(*********************************** G.D S.p.A. - Technical Department ***********************************
============= PROGRAM INFO ============
FOLDER:             TBD
MACHINES INVOLVED:  TBD 

============= DESCRIPTION =============

============= REVISIONS ===============
Date		Version	 	Author      	Description             
----------	-------		------------  	--------------------------------------------
2019/04/24 	0000.00	 	M.Grasso		Creation of the PRG

**********************************************************************************************************)
(*$R
	process_ref := prc;
$*)
PROGRAM csp_main_safety
VAR
	prc:					process;
	prc_path:				STRING;
	
	series_closed_dvr:		BOOL;
	
END_VAR

_read_var_input();

_object_manager();

IF NOT objects_running()
THEN
	RETURN;	
END_IF

_read_process_image();

_mode_manager();

CASE process_get_mode(prc) of
	MODE_ABSENT,
	MODE_INACTIVE:
		RETURN;
	MODE_TEST:
		_handle_process_test();
END_CASE

_set_runtime_properties();

(********************************* BODY *********************************)

(************************************************************************)

_handle_messages();

_write_output();

ACTION _handle_messages:
;
END_ACTION

ACTION _handle_process_test:
;
END_ACTION

ACTION _mode_manager:
IF process_mode_req_is_pending(prc)
THEN
    process_apply_mode_req_first_step(prc);
    CASE process_get_mode(prc) OF
        MODE_TO_ABSENT:
			;
        MODE_TO_INACTIVE:
			;
        MODE_TO_TEST:
			;
        MODE_TO_OPERATIONAL:
			;
    END_CASE
    process_apply_mode_req_second_step(prc);
END_IF
END_ACTION

ACTION _object_manager:
IF objects_initialization()
THEN
	sub_process_init(
		object_name					:= 'csp_main_safety.prc', 
		process						:= csp_main.prc, 
		CONVERSION_this				:= prc);
		
	prc_path 						:= process_get_path(prc);
END_IF

IF objects_running()
THEN
	process_cycle(prc);
END_IF
END_ACTION

ACTION _read_process_image:
	series_closed_dvr := csp_case_main_safety.series_closed_dvr;
END_ACTION

ACTION _read_var_input:
;
END_ACTION

ACTION _set_runtime_properties:
;
END_ACTION

ACTION _write_output:
;
END_ACTION

END_PROGRAM

(* stored: Version 1.1.0.1, ProductVersion 3.1.4024.3
   POU csp_main_safety: Id {0abe4b41-751e-475f-b3c1-2d78dd78ec19}, SpecialFunc None
   Action _handle_messages: Id {a2d2e781-5111-4b8a-bda5-520d47c04e44}
   Action _handle_process_test: Id {23fd720c-e2f9-4b0d-88d2-a815dc7dff6a}
   Action _mode_manager: Id {c48c252e-1912-4389-b805-4aac79ece6b1}
   Action _object_manager: Id {047aa712-0e16-4ce7-896b-bb7e7df91c0f}
   Action _read_process_image: Id {6cc13691-0643-4bbc-8804-31677e2fd356}
   Action _read_var_input: Id {c7f87476-23e2-4bed-9d6f-7ae096d0624a}
   Action _set_runtime_properties: Id {4ff50c29-93bd-44b2-814c-2d8350eb91da}
   Action _write_output: Id {6fb63f4e-fb6b-4932-88d3-609bb4c11c64} *)
